// TwinCAT 3 PLC project ModBusTest
// ProgramVersion: 3.1.4026.9
// libraries:
//   Tc2_ModbusSrv, * (Beckhoff Automation GmbH)
//   Tc2_Standard, * (Beckhoff Automation GmbH)
//   Tc2_System, * (Beckhoff Automation GmbH)
//   Tc3_Module, * (Beckhoff Automation GmbH)
// project tree:
//   GVLs/ GVL.TcGVL
//   / PlcTask.TcTTO
//   POUs/ MAIN.TcPOU
// real-time tasks:
//   TASK PlcTask: cycle T#10ms, priority 20, ADS port 350

CONFIGURATION ModBusTest
    RESOURCE PLC ON TwinCAT3
        TASK PlcTask(INTERVAL := T#10ms, PRIORITY := 20);
        PROGRAM MAIN WITH PlcTask : MAIN;
    END_RESOURCE
END_CONFIGURATION

// ---- GVLs/GVL.TcGVL
{attribute 'qualified_only'}
VAR_GLOBAL
	mb_Input_Coils    		:    ARRAY [0..255] OF BOOL;
	mb_Output_Coils 		:    ARRAY [0..255] OF BOOL;
	mb_Input_Registers 		:    ARRAY [0..255] OF WORD;
	mb_Output_Registers 	:    ARRAY [0..255] OF WORD;
END_VAR

// ---- POUs/MAIN.TcPOU
PROGRAM MAIN
VAR
	b1		:BOOL;
	i1		:INT;
	i2		:INT;
	
	fbADSRead	:ADSREAD;
	fbREdge		:R_TRIG;
	
	bStart		AT %I* :BOOL;
	
END_VAR

FOR i1 := 1 TO 10 BY 1 DO;
	i2:=i2 + 1;
END_FOR

fbADSRead.NETID := '192.168.15.15.1.1';
fbADSRead.PORT := 10500;
fbADSRead.IDXGRP  := 16#2000;
fbADSRead.IDXOFFS := 0;

fbREdge(CLK:=bStart,Q=>);

fbADSRead(
		READ:=fbREdge.Q
		);

END_PROGRAM
